{attribute 'linkalways'} 
{attribute 'no_explicit_call' := 'This FB is a CLASS and must be accessed using methods or properties'}
{attribute 'enable_dynamic_creation'}
FUNCTION_BLOCK _ETcVnPrototypeClusterer EXTENDS EnumDatatypeBase
VAR
	localData : ETcVnPrototypeClusterer;
	activeData : REFERENCE TO ETcVnPrototypeClusterer;
	enumBaseDatatype : _UDINT(localData);
END_VAR

METHOD PRIVATE AddLocalEnumeration
VAR_INPUT
	Enumeration : T_MAXSTRING;
	Value : ETcVnPrototypeClusterer;
END_VAR
AddEnumeration(Enumeration, Value);
END_METHOD

PROPERTY PUBLIC Address : PVOID
GET
Address := ADR(activeData);
END_GET
END_PROPERTY

METHOD PUBLIC ClearReference
VAR_INPUT
END_VAR
activeData REF= localData;
SetBaseDatatypeReference();
END_METHOD

METHOD PUBLIC Clone : I_Datatype
VAR
    pClone : POINTER TO _ETcVnPrototypeClusterer;
END_VAR
pClone := __NEW(_ETcVnPrototypeClusterer(InitialValue := Value));
Clone := pClone^;
END_METHOD

METHOD FB_init : BOOL
VAR_INPUT
	bInitRetains : BOOL; // if TRUE, the retain variables are initialized (warm start / cold start)
	bInCopyCode : BOOL;  // if TRUE, the instance afterwards gets moved into the copy code (online change)
	InitialValue : ETcVnPrototypeClusterer;
END_VAR
localData := InitialValue;
AddBaseDatatype(enumBaseDatatype);
ClearReference();

AddLocalEnumeration('TCVN_PC_NOVELTY_DETECTOR', ETcVnPrototypeClusterer.TCVN_PC_NOVELTY_DETECTOR);
AddLocalEnumeration('TCVN_PC_CLUSTERER', ETcVnPrototypeClusterer.TCVN_PC_CLUSTERER);
END_METHOD

PROPERTY PUBLIC Identifier : T_MAXSTRING
GET
Identifier := 'ETcVnPrototypeClusterer';
END_GET
END_PROPERTY

METHOD IsEnumeratorValueEqual : BOOL
VAR_INPUT
	Enumerator : I_KeyValueForwardEnumerator;
END_VAR
VAR
	storedValue : ETcVnPrototypeClusterer;
END_VAR
IF NOT Enumerator.TryGet(storedValue) THEN
	RETURN;
END_IF

IsEnumeratorValueEqual := storedValue = activeData;
END_METHOD

METHOD PUBLIC MakeReferenceTo
VAR_INPUT
	ReferenceTarget : REFERENCE TO ETcVnPrototypeClusterer;
END_VAR
activeData REF= ReferenceTarget;
SetBaseDatatypeReference();
END_METHOD

METHOD PROTECTED SetBaseDatatypeReference
VAR_INPUT
END_VAR
enumBaseDatatype.MakeReferenceTo(activeData);
END_METHOD

PROPERTY PUBLIC Size : UDINT
GET
Size := SIZEOF(activeData);
END_GET
END_PROPERTY

METHOD TryMakeReferenceTo : BOOL
VAR_INPUT
	Target : I_Datatype;
END_VAR
VAR
	pTargetData : POINTER TO ETcVnPrototypeClusterer;
END_VAR
IF NOT IsEquivalentTo(Target) THEN
	RETURN;
END_IF

pTargetData := Target.Address;
activeData REF= pTargetData^;
SetBaseDatatypeReference();
TryMakeReferenceTo := TRUE;
END_METHOD

PROPERTY PUBLIC Value : ETcVnPrototypeClusterer
GET
Value := activeData;
END_GET
SET
activeData := Value;
END_SET
END_PROPERTY

END_FUNCTION_BLOCK

(* stored: Version 1.1.0.1, ProductVersion 3.1.4024.13
   POU _ETcVnPrototypeClusterer: Id {138d611b-a95a-06ee-06eb-f8aab315d41c}, SpecialFunc None
   Folder Core: Id {ed04411f-75be-0940-285b-e2590a6d37d3}
   Folder Protected: Id {5328203f-cf04-0cac-0a3c-698801aeacd3}
   Folder Customize: Id {37083675-2e5e-0bf4-000a-9c207fd7aa54}
   Folder Constructor: Id {d78fa327-b523-0d78-0083-90921e6d2417}
   Folder Private: Id {3b5796bb-aa84-0df7-0aff-ced346c5c069}
   Folder Protected: Id {f0e0c371-70aa-01b3-018e-06b1722745e3}
   Method AddLocalEnumeration: Id {3ea5117a-1d33-0b52-1cea-c675db4b9957}
   Property Address: Id {244b73d6-a422-0de6-1678-96fc296898c2}
   Get Get: Id {94dd8353-896a-0b46-0945-f09bfb80f265}
   Method ClearReference: Id {183ee3e6-7786-0686-0b62-5fa89bd97e0f}
   Method Clone: Id {c15a772a-5c02-01e6-3674-c3ac53c8d190}
   Method FB_init: Id {bdc02243-4813-0660-175a-05a22a9a5222}
   Property Identifier: Id {266801ce-7c4d-0760-2910-dd1d282fb9ab}
   Get Get: Id {6cbde3db-42af-0d16-12b5-e5d93dee1b5f}
   Method IsEnumeratorValueEqual: Id {8d604112-9dbb-0cee-3d84-f12424b6814b}
   Method MakeReferenceTo: Id {2a3ecfd9-e9c2-00e1-00be-4af15790b016}
   Method SetBaseDatatypeReference: Id {83d80f12-420c-0fa5-2f97-707cfae0f412}
   Property Size: Id {d46202d5-347b-0173-0aa8-7d0d473ce8a3}
   Get Get: Id {06e1296b-d88a-0072-3e1a-02fae97c91dc}
   Method TryMakeReferenceTo: Id {32b3c5a1-147c-087c-00ae-46097de72fd3}
   Property Value: Id {3a0e63f7-b656-052d-357c-f5c85dc22994}
   Get Get: Id {efa80092-5cc5-0fba-00a2-fc41c513fadf}
   Set Set: Id {374be6ed-3b77-0827-1237-0af580fd878c} *)
